{attribute 'linkalways'} 
{attribute 'no_explicit_call' := 'This FB is a CLASS and must be accessed using methods or properties'}
{attribute 'enable_dynamic_creation'}
FUNCTION_BLOCK FINAL MIN_UINT EXTENDS Node
VAR
	in1 : _UINT(0);
	in2 : _UINT(0);
	out : _UINT(0);
END_VAR

METHOD PUBLIC Clone : I_Node
VAR
	pNode : POINTER TO MIN_UINT;
END_VAR
pNode := __NEW(MIN_UINT);
Clone := pNode^;
END_METHOD

METHOD FB_init : BOOL
VAR_INPUT
	bInitRetains : BOOL; // if TRUE, the retain variables are initialized (warm start / cold start)
	bInCopyCode : BOOL;  // if TRUE, the instance afterwards gets moved into the copy code (online change)
END_VAR
AddInput('in1',THIS^.in1);
AddInput('in2',THIS^.in2);
AddOutput('out', THIS^.out);
END_METHOD

METHOD PROTECTED OnExecute
VAR
END_VAR
out.Value := MIN(in1.Value, in2.Value);
END_METHOD

END_FUNCTION_BLOCK

(* stored: Version 1.1.0.1, ProductVersion 3.1.4024.15
   POU MIN_UINT: Id {33c0e12d-44c8-4369-81f5-25b1c8bf8472}, SpecialFunc None
   Folder Constructor: Id {4cb12cda-4d1b-4a93-9d51-a1990beb817e}
   Method Clone: Id {a699b8ad-26ac-4af6-959d-04ced244044a}
   Method FB_init: Id {c81bb069-44c9-4032-992d-e06940b16f48}
   Method OnExecute: Id {c285f69a-7995-4a7c-b66d-585e7217def8} *)
